INTERFACE I_StringLookupINT EXTENDS I_Fallible


METHOD Lookup : INT
VAR_INPUT
    StringToLookup : T_MaxString;
END_VAR
END_METHOD

END_INTERFACE

(* stored: Version 1.1.0.1
   Itf I_StringLookupINT: Id {b48e5a51-e158-43eb-999a-3d2fa3442133}
   Method Lookup: Id {6524db21-4a66-485c-ae51-00a36a3176da} *)
